INTERFACE ITF_Control1 EXTENDS ITF_BaseControlElement

END_INTERFACE

(* stored: Version 1.1.0.1
   Itf ITF_Control1: Id {9b410981-a725-09d5-2d02-18af136f6e58} *)
